{attribute addProperty BoxType "EK1100-0000-0018"}
{attribute addProperty Id "Beckhoff_EL69xxEK1122Beckhoff_EL69xxEK1122_A2B2F2D8162A_0001_EL6900_0000_0016EL6900_F4E3551D16020A_0002_EL6900_0000_0017EL6900_F4E3551D16020A_0003_EL6900_0000_0018EL6900_F4E3551D16020A_0004_EL6900_0000_0019EL6900_F4E3551D16020A_0005_EL6910_0000_0017EL6910_13AA933411214A_0006_EL6910_0000_0018EL6910_13AA933411214A_0007_EL6910_0000_0019EL6910_13AA933411214A_0008_EL6910_0000_0020EL6910_13AA933411214A_0009_EL6930_0000_0016EL6930_F4E3551D16020A_0010_EL6930_0000_0017EL6930_F4E3551D16020A_0011_EL6930_0000_0018EL6930_F4E3551D16020"}
{attribute addProperty CRC "4220474749"}
{attribute addProperty SizeInBites "1584"}
{attribute addProperty SizeInBytes "198"}
TYPE Beckhoff_EL69xx_FB8F557D EXTENDS EK1100_179A0949 :
STRUCT
	{attribute addProperty Name "Beckhoff_EL69xxEK1122"}
	Beckhoff_EL69xxEK1122 : Beckhoff_EL69xxEK1122_A2B2F2D8;
	{attribute addProperty Name "A_0001_EL6900_0000_0016"}
	A_0001_EL6900_0000_0016 : EL6900_F4E3551D;
	{attribute addProperty Name "A_0002_EL6900_0000_0017"}
	A_0002_EL6900_0000_0017 : EL6900_F4E3551D;
	{attribute addProperty Name "A_0003_EL6900_0000_0018"}
	A_0003_EL6900_0000_0018 : EL6900_F4E3551D;
	{attribute addProperty Name "A_0004_EL6900_0000_0019"}
	A_0004_EL6900_0000_0019 : EL6900_F4E3551D;
	{attribute addProperty Name "A_0005_EL6910_0000_0017"}
	A_0005_EL6910_0000_0017 : EL6910_13AA9334;
	{attribute addProperty Name "A_0006_EL6910_0000_0018"}
	A_0006_EL6910_0000_0018 : EL6910_13AA9334;
	{attribute addProperty Name "A_0007_EL6910_0000_0019"}
	A_0007_EL6910_0000_0019 : EL6910_13AA9334;
	{attribute addProperty Name "A_0008_EL6910_0000_0020"}
	A_0008_EL6910_0000_0020 : EL6910_13AA9334;
	{attribute addProperty Name "A_0009_EL6930_0000_0016"}
	A_0009_EL6930_0000_0016 : EL6930_F4E3551D;
	{attribute addProperty Name "A_0010_EL6930_0000_0017"}
	A_0010_EL6930_0000_0017 : EL6930_F4E3551D;
	{attribute addProperty Name "A_0011_EL6930_0000_0018"}
	A_0011_EL6930_0000_0018 : EL6930_F4E3551D;
END_STRUCT
END_TYPE

(* stored: Version 1.2.0.0, ProductVersion 3.1.4024.9
   DUT Beckhoff_EL69xx_FB8F557D: Id {8f58a4a0-472e-4349-941b-30a642841622} *)
